(* PLC project coils_edges, plcc plcc tests 1 *)
(* stored: creationDateTime 2026-09-27T00:00:00 *)

PROGRAM Coils
  VAR
    SetBtn : BOOL;
    ResetBtn : BOOL;
    Latch : BOOL;
    NotLatch : BOOL;
    In : BOOL;
    RisePulse : BOOL;
    FallPulse : BOOL;
    PulseCoil : BOOL;
    DropCoil : BOOL;
    Rises : INT;
  END_VAR
  VAR  (* added by the conversion: wires and edge detectors of the diagram *)
    R_TRIG1 : R_TRIG;
    F_TRIG2 : F_TRIG;
    R_TRIG3 : R_TRIG;
    F_TRIG4 : F_TRIG;
  END_VAR

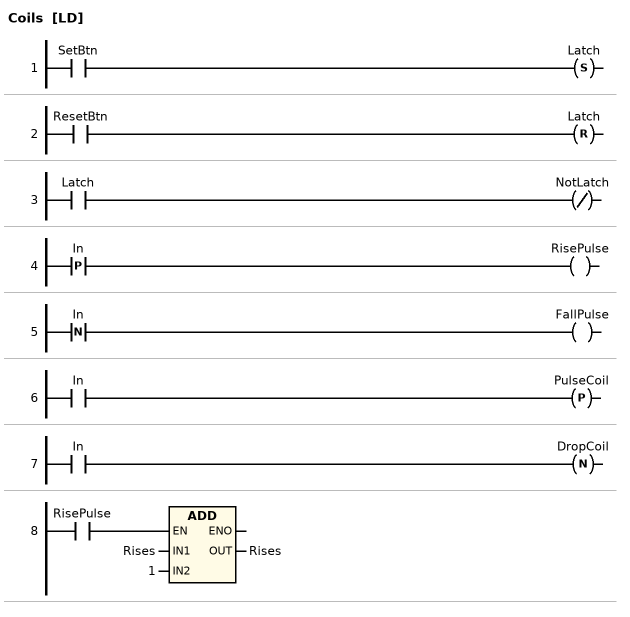
(* LD diagram, written out as Structured Text *)
IF SetBtn THEN Latch := TRUE; END_IF;
IF ResetBtn THEN Latch := FALSE; END_IF;
NotLatch := NOT Latch;
R_TRIG1(CLK := In);
RisePulse := R_TRIG1.Q;
F_TRIG2(CLK := In);
FallPulse := F_TRIG2.Q;
R_TRIG3(CLK := In);
PulseCoil := R_TRIG3.Q;
F_TRIG4(CLK := In);
DropCoil := F_TRIG4.Q;
IF RisePulse THEN Rises := Rises + 1; END_IF;
END_PROGRAM
